PROGRAM otherMachineState
VAR_INPUT
	lightShow:BOOL;
END_VAR
VAR
	inChamberState:UDINT;
	outChamberState:UDINT;
	etchState:UDINT;
	t1:TON;
	rTrig:R_TRIG;
END_VAR

// Chamber State
// Wafer In Chamber State
IF gCtrlMode=ControlMode.eManualCtrMode THEN
	CASE inChamberState OF
		0:
			// 无 Wafer 状态
			IF gWaferMemoryState=0 THEN
				inChamberState:=inChamberState+10;
			END_IF
		10:
			// 实时检测放入晶圆
			IF gICP.I_WaferCheck AND gICP.I_ARMHome THEN
				inChamberState:=inChamberState+10;
			ELSE
				inChamberState:=0;
			END_IF
		20:
			IF gICP.GateDoorExtSensor THEN
				inChamberState:=inChamberState+10;
			ELSE
				inChamberState:=0;
			END_IF
		30:
			IF NOT gICP.I_ARMHome THEN
				inChamberState:=inChamberState+10;
			ELSE
				inChamberState:=20;
			END_IF
		40:
			IF gARMPosition=gICP.ARM.actpos THEN
				inChamberState:=inChamberState+10;
			ELSE
				inChamberState:=20;
			END_IF
		50:
			IF gICP.LiftPinExtSensor THEN// 顶起
				inChamberState:=100;
				gWaferMemoryState:=1;
				ups_CX51X0.Act_Wrtie();
			ELSE
				inChamberState:=200;// 不顶起
				gWaferMemoryState:=0;
				ups_CX51X0.Act_Wrtie();
			END_IF
		100:
			IF ABS( gARMPosition-gICP.ARM.actpos)>1 THEN// 手臂回原
				inChamberState:=inChamberState+10;
			ELSE
				inChamberState:=50;// 手臂静止
			END_IF
		110:
			IF gICP.I_ARMHome THEN
				inChamberState:=0;
			END_IF
			IF gARMPosition=gICP.ARM.actpos THEN
				inChamberState:=40;
			END_IF
		200:
			IF ABS( gARMPosition-gICP.ARM.actpos)>1 THEN// 手臂回原
				inChamberState:=inChamberState+10;
			ELSE
				inChamberState:=50;// 手臂静止
			END_IF
		210:
			IF gICP.I_ARMHome THEN
				inChamberState:=0;
			END_IF
			IF gARMPosition=gICP.ARM.actpos THEN
				inChamberState:=40;
			END_IF
	END_CASE
	
	CASE outChamberState OF
		0:
			// 有 Wafer 状态
			IF gWaferMemoryState=1 THEN
				outChamberState:=outChamberState+10;
			END_IF
		10:
			IF gICP.GateDoorExtSensor AND gARMPosition=gICP.ARM.actpos THEN
				outChamberState:=outChamberState+10;
			ELSE
				outChamberState:=0;
			END_IF
		20:
			IF gICP.LiftPinExtSensor THEN
				outChamberState:=outChamberState+10;
			END_IF
		30:
			IF gICP.LiftPinRetSensor THEN
				gWaferMemoryState:=0;
				ups_CX51X0.Act_Wrtie();
				outChamberState:=outChamberState+10;
			ELSE
				IF ABS( gARMPosition-gICP.ARM.actpos)>1 THEN
					outChamberState:=0;
				END_IF
			END_IF	
		40:
			IF gICP.I_ARMHome THEN
				outChamberState:=0;
			END_IF
			IF gICP.LiftPinExtSensor THEN
				gWaferMemoryState:=1;
				ups_CX51X0.Act_Wrtie();
				outChamberState:=20;
			END_IF
	END_CASE
END_IF
t1(IN:=gWaferMemoryState=1 AND NOT t1.Q,PT:=T#0.5S);
IF t1.Q THEN
	lightShow:=NOT lightShow;
END_IF
IF gWaferMemoryState=0 THEN
	lightShow:=FALSE;
END_IF

IF S_ActuatorRecoveryPOU.busy OR MainPOU.busy OR S_ChamberLLVent.busy OR S_Etching.busy OR S_LoadLockPumping.busy OR S_LoadLockVent.busy OR
	S_LoadWafer.busy OR S_MachinePumping.busy OR S_MachineVent.busy OR S_RoughPumping.busy OR S_UnLoadWafer.busy OR S_WaferCheckPOU.busy OR
	S_PDVSafeCtr.busy THEN
	gSPOUBusy:=TRUE;
ELSE
	gSPOUBusy:=FALSE;
	gShowPOURunLog:=FALSE;
END_IF
gRunningLog.clearShowInfo:=FALSE;
rTrig(CLK:=gSPOUBusy);
IF rTrig.Q THEN
	gRunningLog.clearShowInfo:=TRUE;
	gShowPOURunLog:=TRUE;
END_IF
IF NOT gSPOUBusy THEN
	IF gICP.TBGauge.outputValue<400 THEN
		gRoughRemainTMPCanOpen:=TRUE;
	ELSE
		gRoughRemainTMPCanOpen:=FALSE;
	END_IF
ELSE
	IF gICP.TBGauge.outputValue>400 THEN
		gRoughRemainTMPCanOpen:=FALSE;
	END_IF
END_IF

IF ABS(gICP.MFC1.setFlow-gICP.MFC1.actflow)>gMFCMonitParLimit OR  ABS(gICP.MFC2.setFlow-gICP.MFC2.actflow)>gMFCMonitParLimit OR  ABS(gICP.MFC3.setFlow-gICP.MFC3.actflow)>gMFCMonitParLimit 
	OR  ABS(gICP.MFC4.setFlow-gICP.MFC4.actflow)>gMFCMonitParLimit OR  ABS(gICP.MFC5.setFlow-gICP.MFC5.actflow)>gMFCMonitParLimit OR  ABS(gICP.MFC6.setFlow-gICP.MFC6.actflow)>gMFCMonitParLimit 
	OR  ABS(gICP.MFC7.setFlow-gICP.MFC7.actflow)>gMFCMonitParLimit OR  ABS(gICP.MFC8.setFlow-gICP.MFC8.actflow)>gMFCMonitParLimit OR  ABS(gICP.MFC9.setFlow-gICP.MFC9.actflow)>gMFCMonitParLimit  THEN
	gICP.S_MFCMonitFlowNotZero:=TRUE;
ELSE
	gICP.S_MFCMonitFlowNotZero:=FALSE;
END_IF

METHOD RecipeInputCheck : BOOL
VAR_INPUT
	numMax:INT;
END_VAR
VAR
	start:INT:=1;
	i:INT;
END_VAR
FOR start:=1 TO numMax DO
	IF len(gRecipeViewData[start].mfc1)>0 THEN
		FOR i:=0 TO LEN(gRecipeViewData[start].mfc1)-1 DO
			gLog.append(BYTE_TO_STRING(gRecipeViewData[start].mfc1[i]));
		END_FOR
	END_IF
END_FOR
END_METHOD

END_PROGRAM

(* stored: Version 1.1.0.1, ProductVersion 3.1.4024.12
   POU otherMachineState: Id {fca6f4e4-5ae4-444c-9ed7-235dd6d71b99}, SpecialFunc None
   Method RecipeInputCheck: Id {9fd3f976-ea6b-456c-9f7f-de0e99b12e4d} *)
